(* IEC 61131-3 sources: robocpp/validation/corpus/c-parity, 1 file *)

(* ---- counter_codegen.st ---- *)
(* validation: feature=backend.generated-c clause=backend.c program=CounterDemo *)
PROGRAM CounterDemo
VAR
    Count : INT := 0;
    Limit : INT := 3;
    Done : BOOL := FALSE;
END_VAR

IF Count < Limit THEN
    Count := Count + 1;
ELSE
    Done := TRUE;
END_IF;
END_PROGRAM
